// TIA Portal V16 export
// export: Created 2021-11-12T13:32:39.4963653Z, ExportSetting WithDefaults, DisplayName Totally Integrated Automation Portal, DisplayVersion V16 Update 3, DisplayName TIA Portal Version Control Interface, DisplayVersion V16 Update 2, DisplayName TIA Portal Openness, DisplayVersion V16 Update 3, DisplayName SINAMICS Startdrive Advanced, DisplayVersion V16 Update 5, DisplayName SINAMICS Startdrive G130, G150, S120, S150, SINAMICS MV, S210, DisplayVersion V16 Update 5, DisplayName SINAMICS Startdrive G110M, G120, G120C, G120D, G120P, G115D, DisplayVersion V16 Update 5, DisplayName STEP 7 Professional, DisplayVersion V16 Update 3, DisplayName STEP 7 Safety, DisplayVersion V16, DisplayName WinCC UA Professional, DisplayVersion V16 Update 3
FUNCTION_BLOCK "Station2R2"   // FB19, LAD
{ S7_Optimized_Access := 'TRUE' }
VERSION : 0.1
// stored: AutoNumber true, IsIECCheckEnabled false, IsRetainMemResEnabled false, MemoryReserve 100, SetENOAutomatically false, UDAEnableTagReadback false
   VAR
      SF_RO01_Timeout : "STD_DI_Mon";
      SF_RO01_LubStartErr { S7_SetPoint := 'True'} : "STD_DI_Mon";
      "SF_CM01-BL01_Wrn" { S7_SetPoint := 'True'} : "STD_DI_Mon";
      "SF_CM01-BL01_Err" { S7_SetPoint := 'True'} : "STD_DI_Mon";
      SF_RO01 { S7_SetPoint := 'True'} : "STD_RobotABB";
      SF_RC01 : "STD_DriveRobotABB";
      SS_Edge { S7_SetPoint := 'True'} : Array[0..16] of Bool;
      SB1ReqServPos { ExternalAccessible := 'False'; ExternalVisible := 'False'; ExternalWritable := 'False'} : Bool;   // Request to go to/from service position
      SB1ReqToolchange : Bool;   // Go to position for change tool request
      SB1ReqFlush : Bool;   // Request to flash tool
      SB1ReqFlushAux { ExternalAccessible := 'False'; ExternalVisible := 'False'; ExternalWritable := 'False'} : Bool;   // Manual (HW button) request to flush
      SB1ReqSprayMan : Bool;   // Manual (HW button) request to spray
      SB1ReqSprayManAux { ExternalAccessible := 'False'; ExternalVisible := 'False'; ExternalWritable := 'False'} : Bool;   // Manual (HW button) request to spray
      SB1CycleAutostop : Bool;   // Cycle autostop command
      SB1RobotInitialized : Bool;   // SB1RobotInitialized
   END_VAR
   VAR_TEMP
      TS_RC01 : "UDT_DriveRobotABBControl";   // Robot RO01 control
      TS_RO01 : "UDT_RobotABBControl";   // Robot RO01 control
      TB1PwrOK : Bool;   // Power for this station is OK
      TB1CtrlRun : Bool;   // Robot controller is running in automat
      TB1HomePos : Bool;   // Request to go to home position
      TB1MoveOutPress : Bool;   // Move robout out of press
      TB1SprayInPress : Bool;   // Spray into press
      TB1SprayOutPress : Bool;   // Spray out off press
      TB1SprayMan : Bool;   // Spray manually both ways
      TB1Flush : Bool;   // Flush tool
      TB1MoveToStandBy : Bool;   // From home to StandBy
      TB1PressFree : Bool;   // positions in press are free
      TB1PartsBefore : Bool;   // Parts in zone before robot
   END_VAR
   VAR CONSTANT
      CI_JobHome : UInt := 1;   // Go home
      CI_JobService : UInt := 2;   // Go service
      CI_JobToolchange : UInt := 3;   // Go to position for change tool
      CI_JobMoveOutPress : UInt := 11;   // Move out of the press
      CI_JobStandBy : UInt := 12;   // From home to StandBy
      CI_JobSprayIntoPress : UInt := 101;   // Spray into the press
      CI_JobSprayOutPress : UInt := 102;   // Spray out of the press
      CI_JobSprayMan : UInt := 110;   // Spray manually both ways
      CI_JobFlushTool : UInt := 200;   // Flush
   END_VAR
   VAR_TEMP   // added for the SCL form of the ladder/FBD networks
      _w1 : Bool;
      _w2 : Bool;
      _w3 : Bool;
      _w4 : Bool;
   END_VAR
BEGIN

REGION Network 1: Clear temporary variables
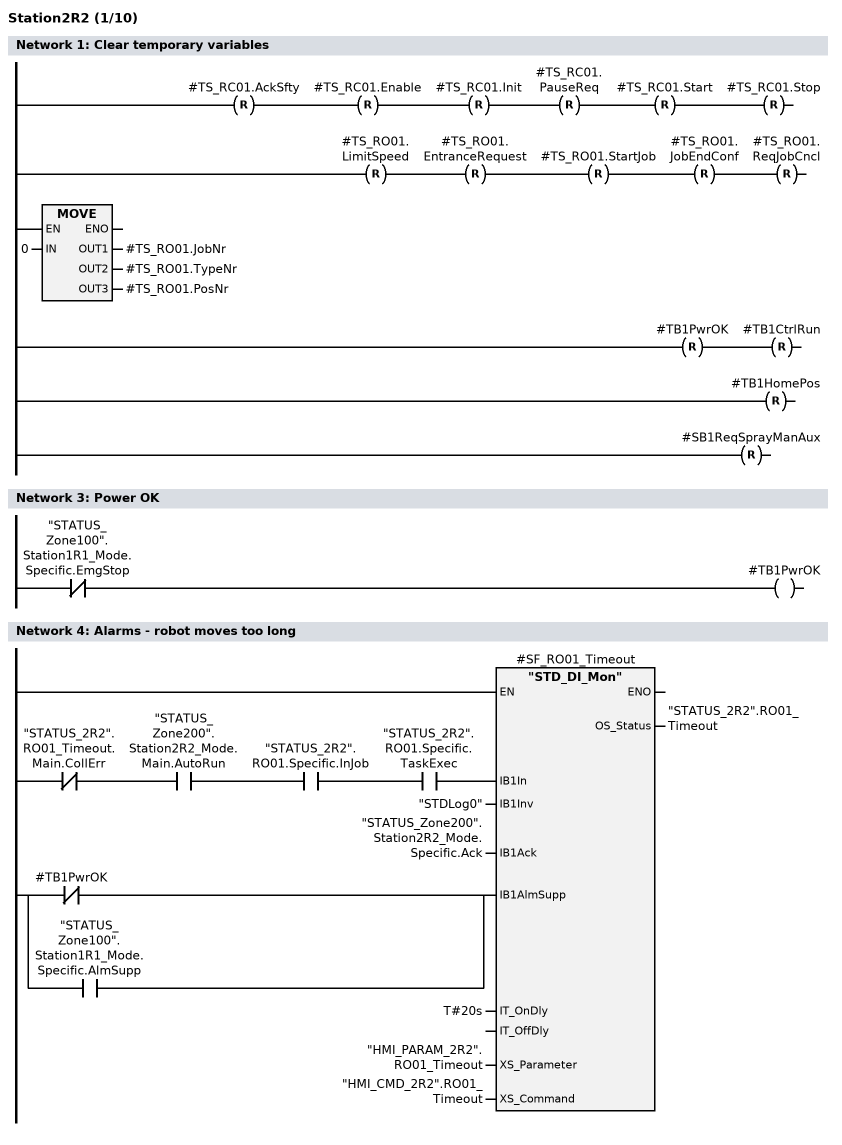
   RUNG wire#powerrail
      R_Coil( #TS_RC01.AckSfty )
      R_Coil( #TS_RC01.Enable )
      R_Coil( #TS_RC01.Init )
      R_Coil( #TS_RC01.PauseReq )
      R_Coil( #TS_RC01.Start )
      R_Coil( #TS_RC01.Stop )
   END_RUNG
   RUNG wire#powerrail
      R_Coil( #TS_RO01.LimitSpeed )
      R_Coil( #TS_RO01.EntranceRequest )
      R_Coil( #TS_RO01.StartJob )
      R_Coil( #TS_RO01.JobEndConf )
      R_Coil( #TS_RO01.ReqJobCncl )
   END_RUNG
   RUNG wire#powerrail
      Move(in := 0, out1 => #TS_RO01.JobNr, out2 => #TS_RO01.TypeNr, out3 => #TS_RO01.PosNr)
   END_RUNG
   RUNG wire#powerrail
      R_Coil( #TB1PwrOK )
      R_Coil( #TB1CtrlRun )
   END_RUNG
   RUNG wire#powerrail
      R_Coil( #TB1HomePos )
   END_RUNG
   RUNG wire#powerrail
      R_Coil( #SB1ReqSprayManAux )
   END_RUNG
   // the same network as SCL:
   #TS_RC01.AckSfty := FALSE;
   #TS_RC01.Enable := FALSE;
   #TS_RC01.Init := FALSE;
   #TS_RC01.PauseReq := FALSE;
   #TS_RC01.Start := FALSE;
   #TS_RC01.Stop := FALSE;
   #TS_RO01.LimitSpeed := FALSE;
   #TS_RO01.EntranceRequest := FALSE;
   #TS_RO01.StartJob := FALSE;
   #TS_RO01.JobEndConf := FALSE;
   #TS_RO01.ReqJobCncl := FALSE;
   #TS_RO01.JobNr := 0;
   #TS_RO01.TypeNr := 0;
   #TS_RO01.PosNr := 0;
   #TB1PwrOK := FALSE;
   #TB1CtrlRun := FALSE;
   #TB1HomePos := FALSE;
   #SB1ReqSprayManAux := FALSE;
END_REGION

REGION Network 2: *************** Alarms ***************
END_REGION

REGION Network 3: Power OK
   RUNG wire#powerrail
      I_Contact( "STATUS_Zone100".Station1R1_Mode.Specific.EmgStop )
      Coil( #TB1PwrOK )
   END_RUNG
   // the same network as SCL:
   #TB1PwrOK := NOT "STATUS_Zone100".Station1R1_Mode.Specific.EmgStop;
END_REGION

REGION Network 4: Alarms - robot moves too long
   RUNG wire#powerrail
      #SF_RO01_Timeout(IB1In := wire#w1, IB1AlmSupp := wire#w2, IB1Inv := "STDLog0", IB1Ack := "STATUS_Zone200".Station2R2_Mode.Specific.Ack, IT_OnDly := T#20s, IT_OffDly :=, XS_Parameter := "HMI_PARAM_2R2".RO01_Timeout, XS_Command := "HMI_CMD_2R2".RO01_Timeout, OS_Status => "STATUS_2R2".RO01_Timeout)
   END_RUNG
   RUNG wire#powerrail
      I_Contact( "STATUS_2R2".RO01_Timeout.Main.CollErr )
      Contact( "STATUS_Zone200".Station2R2_Mode.Main.AutoRun )
      Contact( "STATUS_2R2".RO01.Specific.InJob )
      Contact( "STATUS_2R2".RO01.Specific.TaskExec )
   END_RUNG wire#w1
   RUNG wire#powerrail
      I_Contact( #TB1PwrOK )
   END_RUNG wire#w2
   RUNG wire#powerrail
      Contact( "STATUS_Zone100".Station1R1_Mode.Specific.AlmSupp )
   END_RUNG wire#w2
   // the same network as SCL:
   #SF_RO01_Timeout(IB1In := NOT "STATUS_2R2".RO01_Timeout.Main.CollErr AND "STATUS_Zone200".Station2R2_Mode.Main.AutoRun AND "STATUS_2R2".RO01.Specific.InJob AND "STATUS_2R2".RO01.Specific.TaskExec,   // "STD_DI_Mon"
                    IB1Inv := "STDLog0",
                    IB1Ack := "STATUS_Zone200".Station2R2_Mode.Specific.Ack,
                    IB1AlmSupp := NOT #TB1PwrOK OR "STATUS_Zone100".Station1R1_Mode.Specific.AlmSupp,
                    IT_OnDly := T#20s,
                    XS_Parameter := "HMI_PARAM_2R2".RO01_Timeout,
                    XS_Command := "HMI_CMD_2R2".RO01_Timeout,
                    OS_Status => "STATUS_2R2".RO01_Timeout);
END_REGION

REGION Network 5: Alarm - robot did not move into the press machine
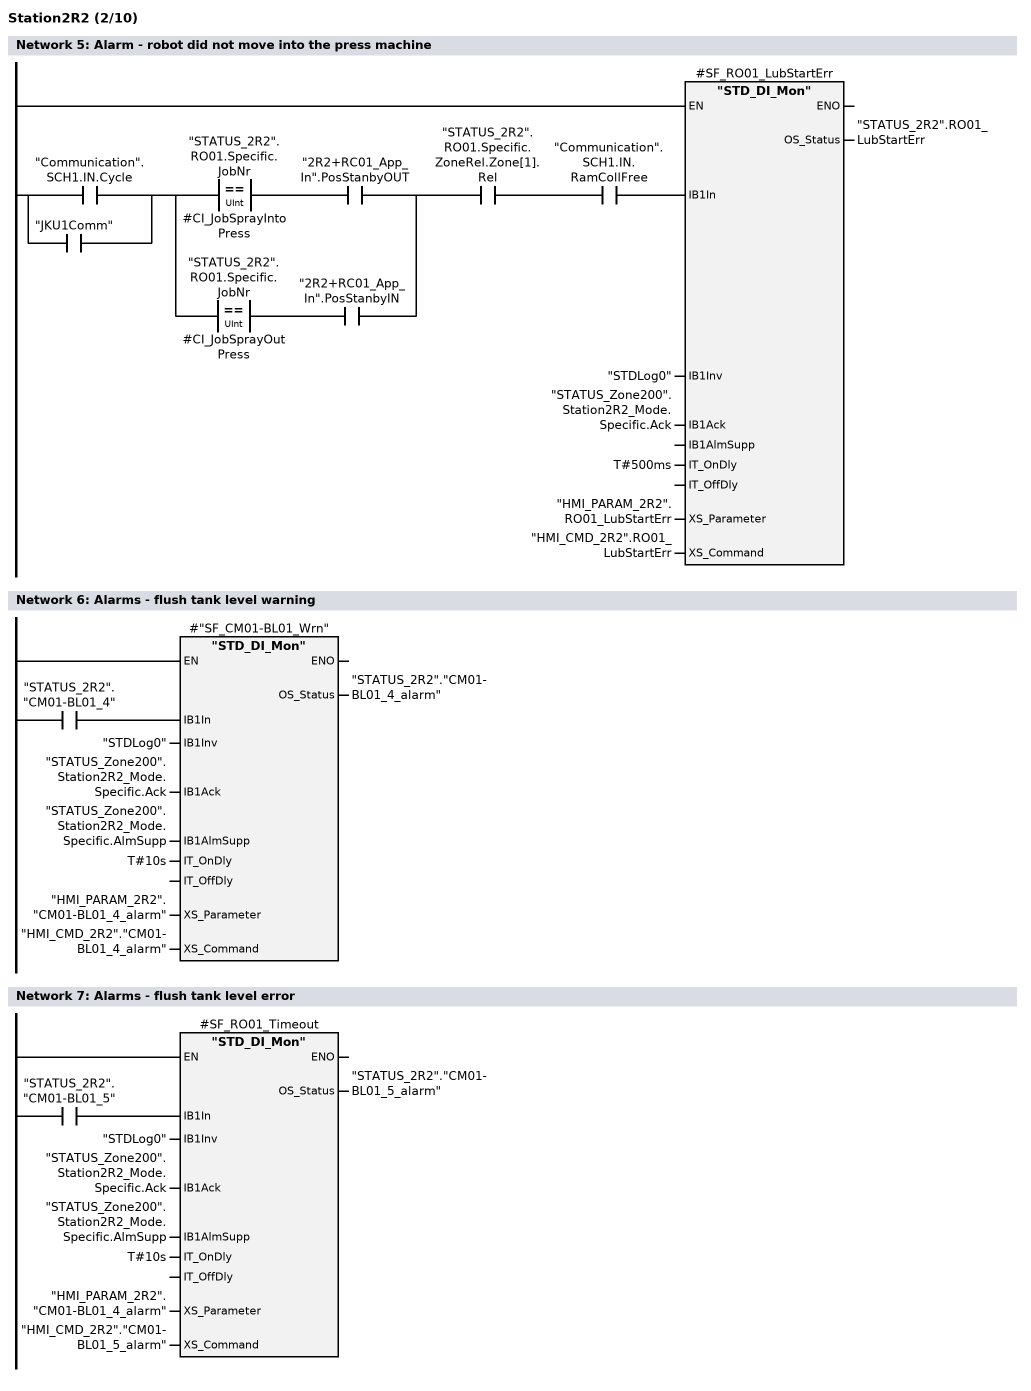
   RUNG wire#powerrail
      #SF_RO01_LubStartErr(IB1In := wire#w3, IB1Inv := "STDLog0", IB1Ack := "STATUS_Zone200".Station2R2_Mode.Specific.Ack, IB1AlmSupp :=, IT_OnDly := T#500ms, IT_OffDly :=, XS_Parameter := "HMI_PARAM_2R2".RO01_LubStartErr, XS_Command := "HMI_CMD_2R2".RO01_LubStartErr, OS_Status => "STATUS_2R2".RO01_LubStartErr)
   END_RUNG
   RUNG wire#powerrail
      Contact( "Communication".SCH1.IN.Cycle )
      wire#w1
      { S7_Templates := "SrcType := UInt" } EQ_Contact(in1 := "STATUS_2R2".RO01.Specific.JobNr, in2 := #CI_JobSprayIntoPress)
      Contact( "2R2+RC01_App_In".PosStanbyOUT )
      wire#w2
      Contact( "STATUS_2R2".RO01.Specific.ZoneRel.Zone[1].Rel )
      Contact( "Communication".SCH1.IN.RamCollFree )
   END_RUNG wire#w3
   RUNG wire#powerrail
      Contact( "JKU1Comm" )
   END_RUNG wire#w1
   RUNG wire#w1
      { S7_Templates := "SrcType := UInt" } EQ_Contact(in1 := "STATUS_2R2".RO01.Specific.JobNr, in2 := #CI_JobSprayOutPress)
      Contact( "2R2+RC01_App_In".PosStanbyIN )
   END_RUNG wire#w2
   // the same network as SCL:
   #SF_RO01_LubStartErr(IB1In := ("Communication".SCH1.IN.Cycle OR "JKU1Comm") AND ((("STATUS_2R2".RO01.Specific.JobNr = #CI_JobSprayIntoPress) AND "2R2+RC01_App_In".PosStanbyOUT) OR (("STATUS_2R2".RO01.Specific.JobNr = #CI_JobSprayOutPress) AND "2R2+RC01_App_In".PosStanbyIN)) AND "STATUS_2R2".RO01.Specific.ZoneRel.Zone[1].Rel AND "Communication".SCH1.IN.RamCollFree,   // "STD_DI_Mon"
                        IB1Inv := "STDLog0",
                        IB1Ack := "STATUS_Zone200".Station2R2_Mode.Specific.Ack,
                        IT_OnDly := T#500ms,
                        XS_Parameter := "HMI_PARAM_2R2".RO01_LubStartErr,
                        XS_Command := "HMI_CMD_2R2".RO01_LubStartErr,
                        OS_Status => "STATUS_2R2".RO01_LubStartErr);
END_REGION

REGION Network 6: Alarms - flush tank level warning
   RUNG wire#powerrail
      #"SF_CM01-BL01_Wrn"(IB1In := wire#w1, IB1Inv := "STDLog0", IB1Ack := "STATUS_Zone200".Station2R2_Mode.Specific.Ack, IB1AlmSupp := "STATUS_Zone200".Station2R2_Mode.Specific.AlmSupp, IT_OnDly := T#10s, IT_OffDly :=, XS_Parameter := "HMI_PARAM_2R2"."CM01-BL01_4_alarm", XS_Command := "HMI_CMD_2R2"."CM01-BL01_4_alarm", OS_Status => "STATUS_2R2"."CM01-BL01_4_alarm")
   END_RUNG
   RUNG wire#powerrail
      Contact( "STATUS_2R2"."CM01-BL01_4" )
   END_RUNG wire#w1
   // the same network as SCL:
   #"SF_CM01-BL01_Wrn"(IB1In := "STATUS_2R2"."CM01-BL01_4",   // "STD_DI_Mon"
                       IB1Inv := "STDLog0",
                       IB1Ack := "STATUS_Zone200".Station2R2_Mode.Specific.Ack,
                       IB1AlmSupp := "STATUS_Zone200".Station2R2_Mode.Specific.AlmSupp,
                       IT_OnDly := T#10s,
                       XS_Parameter := "HMI_PARAM_2R2"."CM01-BL01_4_alarm",
                       XS_Command := "HMI_CMD_2R2"."CM01-BL01_4_alarm",
                       OS_Status => "STATUS_2R2"."CM01-BL01_4_alarm");
END_REGION

REGION Network 7: Alarms - flush tank level error
   RUNG wire#powerrail
      #SF_RO01_Timeout(IB1In := wire#w1, IB1Inv := "STDLog0", IB1Ack := "STATUS_Zone200".Station2R2_Mode.Specific.Ack, IB1AlmSupp := "STATUS_Zone200".Station2R2_Mode.Specific.AlmSupp, IT_OnDly := T#10s, IT_OffDly :=, XS_Parameter := "HMI_PARAM_2R2"."CM01-BL01_4_alarm", XS_Command := "HMI_CMD_2R2"."CM01-BL01_5_alarm", OS_Status => "STATUS_2R2"."CM01-BL01_5_alarm")
   END_RUNG
   RUNG wire#powerrail
      Contact( "STATUS_2R2"."CM01-BL01_5" )
   END_RUNG wire#w1
   // the same network as SCL:
   #SF_RO01_Timeout(IB1In := "STATUS_2R2"."CM01-BL01_5",   // "STD_DI_Mon"
                    IB1Inv := "STDLog0",
                    IB1Ack := "STATUS_Zone200".Station2R2_Mode.Specific.Ack,
                    IB1AlmSupp := "STATUS_Zone200".Station2R2_Mode.Specific.AlmSupp,
                    IT_OnDly := T#10s,
                    XS_Parameter := "HMI_PARAM_2R2"."CM01-BL01_4_alarm",
                    XS_Command := "HMI_CMD_2R2"."CM01-BL01_5_alarm",
                    OS_Status => "STATUS_2R2"."CM01-BL01_5_alarm");
END_REGION

REGION Network 8: *************** Controller RC01 ***************
END_REGION

REGION Network 9: RC01 - control
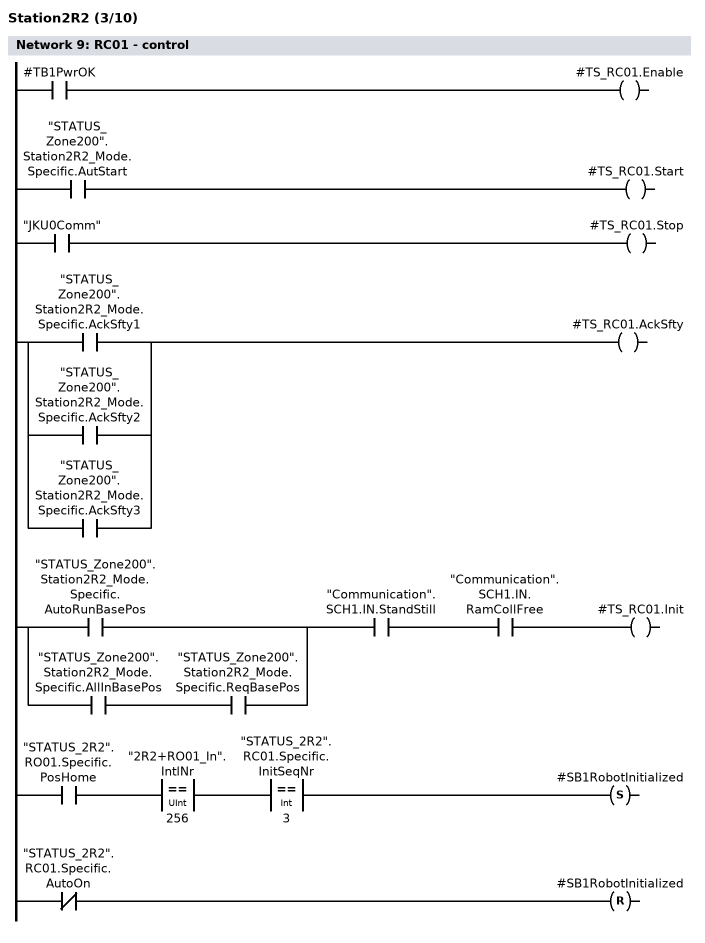
   RUNG wire#powerrail
      Contact( #TB1PwrOK )
      Coil( #TS_RC01.Enable )
   END_RUNG
   RUNG wire#powerrail
      Contact( "STATUS_Zone200".Station2R2_Mode.Specific.AutStart )
      Coil( #TS_RC01.Start )
   END_RUNG
   RUNG wire#powerrail
      Contact( "JKU0Comm" )
      Coil( #TS_RC01.Stop )
   END_RUNG
   RUNG wire#powerrail
      Contact( "STATUS_Zone200".Station2R2_Mode.Specific.AckSfty1 )
      wire#w1
      Coil( #TS_RC01.AckSfty )
   END_RUNG
   RUNG wire#powerrail
      Contact( "STATUS_Zone200".Station2R2_Mode.Specific.AckSfty2 )
   END_RUNG wire#w1
   RUNG wire#powerrail
      Contact( "STATUS_Zone200".Station2R2_Mode.Specific.AckSfty3 )
   END_RUNG wire#w1
   RUNG wire#powerrail
      Contact( "STATUS_Zone200".Station2R2_Mode.Specific.AutoRunBasePos )
      wire#w2
      Contact( "Communication".SCH1.IN.StandStill )
      Contact( "Communication".SCH1.IN.RamCollFree )
      Coil( #TS_RC01.Init )
   END_RUNG
   RUNG wire#powerrail
      Contact( "STATUS_Zone200".Station2R2_Mode.Specific.AllInBasePos )
      Contact( "STATUS_Zone200".Station2R2_Mode.Specific.ReqBasePos )
   END_RUNG wire#w2
   RUNG wire#powerrail
      Contact( "STATUS_2R2".RO01.Specific.PosHome )
      { S7_Templates := "SrcType := UInt" } EQ_Contact(in1 := "2R2+RO01_In".IntlNr, in2 := 256)
      { S7_Templates := "SrcType := Int" } EQ_Contact(in1 := "STATUS_2R2".RC01.Specific.InitSeqNr, in2 := 3)
      S_Coil( #SB1RobotInitialized )
   END_RUNG
   RUNG wire#powerrail
      I_Contact( "STATUS_2R2".RC01.Specific.AutoOn )
      R_Coil( #SB1RobotInitialized )
   END_RUNG
   // the same network as SCL:
   #TS_RC01.Enable := #TB1PwrOK;
   #TS_RC01.Start := "STATUS_Zone200".Station2R2_Mode.Specific.AutStart;
   #TS_RC01.Stop := "JKU0Comm";
   #TS_RC01.AckSfty := "STATUS_Zone200".Station2R2_Mode.Specific.AckSfty1 OR "STATUS_Zone200".Station2R2_Mode.Specific.AckSfty2 OR "STATUS_Zone200".Station2R2_Mode.Specific.AckSfty3;
   #TS_RC01.Init := ("STATUS_Zone200".Station2R2_Mode.Specific.AutoRunBasePos OR ("STATUS_Zone200".Station2R2_Mode.Specific.AllInBasePos AND "STATUS_Zone200".Station2R2_Mode.Specific.ReqBasePos)) AND "Communication".SCH1.IN.StandStill AND "Communication".SCH1.IN.RamCollFree;
   IF "STATUS_2R2".RO01.Specific.PosHome AND ("2R2+RO01_In".IntlNr = 256) AND ("STATUS_2R2".RC01.Specific.InitSeqNr = 3) THEN
       #SB1RobotInitialized := TRUE;
   END_IF;
   IF NOT "STATUS_2R2".RC01.Specific.AutoOn THEN #SB1RobotInitialized := FALSE; END_IF;
END_REGION

REGION Network 10: RC01 - request to pause robots jobs
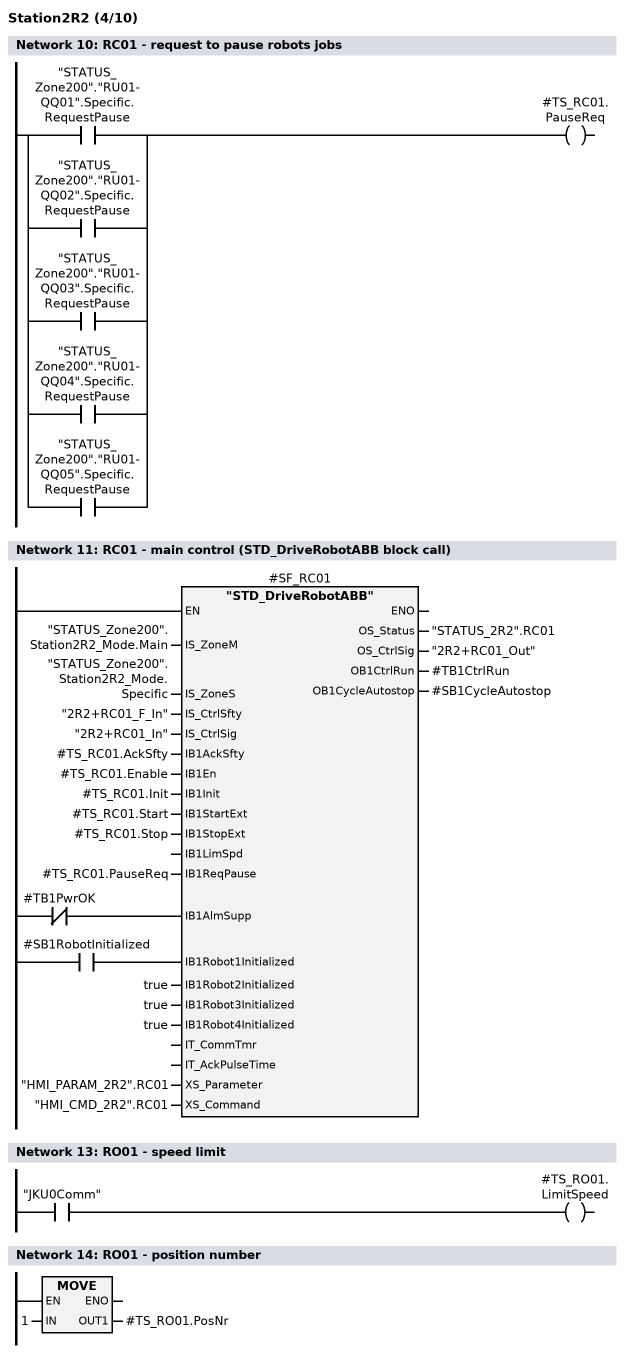
   RUNG wire#powerrail
      Contact( "STATUS_Zone200"."RU01-QQ01".Specific.RequestPause )
      wire#w1
      Coil( #TS_RC01.PauseReq )
   END_RUNG
   RUNG wire#powerrail
      Contact( "STATUS_Zone200"."RU01-QQ02".Specific.RequestPause )
   END_RUNG wire#w1
   RUNG wire#powerrail
      Contact( "STATUS_Zone200"."RU01-QQ03".Specific.RequestPause )
   END_RUNG wire#w1
   RUNG wire#powerrail
      Contact( "STATUS_Zone200"."RU01-QQ04".Specific.RequestPause )
   END_RUNG wire#w1
   RUNG wire#powerrail
      Contact( "STATUS_Zone200"."RU01-QQ05".Specific.RequestPause )
   END_RUNG wire#w1
   // the same network as SCL:
   #TS_RC01.PauseReq := "STATUS_Zone200"."RU01-QQ01".Specific.RequestPause OR "STATUS_Zone200"."RU01-QQ02".Specific.RequestPause OR "STATUS_Zone200"."RU01-QQ03".Specific.RequestPause OR "STATUS_Zone200"."RU01-QQ04".Specific.RequestPause OR "STATUS_Zone200"."RU01-QQ05".Specific.RequestPause;
END_REGION

REGION Network 11: RC01 - main control (STD_DriveRobotABB block call)
   RUNG wire#powerrail
      #SF_RC01(IB1AlmSupp := wire#w1, IB1Robot1Initialized := wire#w2, IS_ZoneM := "STATUS_Zone200".Station2R2_Mode.Main, IS_ZoneS := "STATUS_Zone200".Station2R2_Mode.Specific, IS_CtrlSfty := "2R2+RC01_F_In", IS_CtrlSig := "2R2+RC01_In", IB1AckSfty := #TS_RC01.AckSfty, IB1En := #TS_RC01.Enable, IB1Init := #TS_RC01.Init, IB1StartExt := #TS_RC01.Start, IB1StopExt := #TS_RC01.Stop, IB1LimSpd :=, IB1ReqPause := #TS_RC01.PauseReq, IB1Robot2Initialized := true, IB1Robot3Initialized := true, IB1Robot4Initialized := true, IT_CommTmr :=, IT_AckPulseTime :=, XS_Parameter := "HMI_PARAM_2R2".RC01, XS_Command := "HMI_CMD_2R2".RC01, OS_Status => "STATUS_2R2".RC01, OS_CtrlSig => "2R2+RC01_Out", OB1CtrlRun => #TB1CtrlRun, OB1CycleAutostop => #SB1CycleAutostop)
   END_RUNG
   RUNG wire#powerrail
      I_Contact( #TB1PwrOK )
   END_RUNG wire#w1
   RUNG wire#powerrail
      Contact( #SB1RobotInitialized )
   END_RUNG wire#w2
   // the same network as SCL:
   #SF_RC01(IS_ZoneM := "STATUS_Zone200".Station2R2_Mode.Main,   // "STD_DriveRobotABB"
            IS_ZoneS := "STATUS_Zone200".Station2R2_Mode.Specific,
            IS_CtrlSfty := "2R2+RC01_F_In",
            IS_CtrlSig := "2R2+RC01_In",
            IB1AckSfty := #TS_RC01.AckSfty,
            IB1En := #TS_RC01.Enable,
            IB1Init := #TS_RC01.Init,
            IB1StartExt := #TS_RC01.Start,
            IB1StopExt := #TS_RC01.Stop,
            IB1ReqPause := #TS_RC01.PauseReq,
            IB1AlmSupp := NOT #TB1PwrOK,
            IB1Robot1Initialized := #SB1RobotInitialized,
            IB1Robot2Initialized := true,
            IB1Robot3Initialized := true,
            IB1Robot4Initialized := true,
            XS_Parameter := "HMI_PARAM_2R2".RC01,
            XS_Command := "HMI_CMD_2R2".RC01,
            OS_Status => "STATUS_2R2".RC01,
            OS_CtrlSig => "2R2+RC01_Out",
            OB1CtrlRun => #TB1CtrlRun,
            OB1CycleAutostop => #SB1CycleAutostop);
END_REGION

REGION Network 12: *************** Robot RO01 ***************
END_REGION

REGION Network 13: RO01 - speed limit
   RUNG wire#powerrail
      Contact( "JKU0Comm" )
      Coil( #TS_RO01.LimitSpeed )
   END_RUNG
   // the same network as SCL:
   #TS_RO01.LimitSpeed := "JKU0Comm";
END_REGION

REGION Network 14: RO01 - position number
   RUNG wire#powerrail
      Move(in := 1, out1 => #TS_RO01.PosNr)
   END_RUNG
   // the same network as SCL:
   #TS_RO01.PosNr := 1;
END_REGION

REGION Network 15: RO01 - confirm end of job
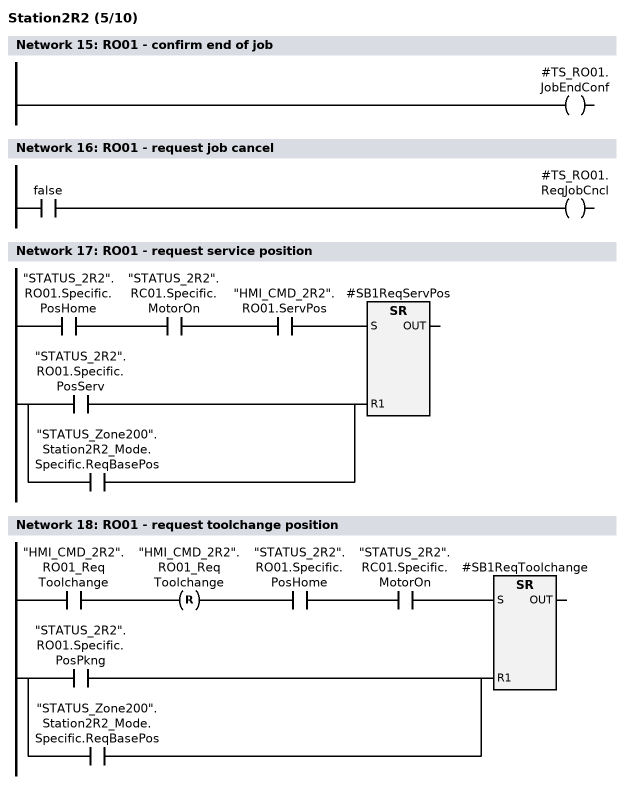
   RUNG wire#powerrail
      Coil( #TS_RO01.JobEndConf )
   END_RUNG
   // the same network as SCL:
   #TS_RO01.JobEndConf := TRUE;
END_REGION

REGION Network 16: RO01 - request job cancel
   RUNG wire#powerrail
      Contact( false )
      Coil( #TS_RO01.ReqJobCncl )
   END_RUNG
   // the same network as SCL:
   #TS_RO01.ReqJobCncl := false;
END_REGION

REGION Network 17: RO01 - request service position
   RUNG wire#powerrail
      Contact( "STATUS_2R2".RO01.Specific.PosHome )
      Contact( "STATUS_2R2".RC01.Specific.MotorOn )
      Contact( "HMI_CMD_2R2".RO01.ServPos )
      S_SR(operand := #SB1ReqServPos, r1 := wire#w1)
   END_RUNG
   RUNG wire#powerrail
      Contact( "STATUS_2R2".RO01.Specific.PosServ )
   END_RUNG wire#w1
   RUNG wire#powerrail
      Contact( "STATUS_Zone200".Station2R2_Mode.Specific.ReqBasePos )
   END_RUNG wire#w1
   // the same network as SCL:
   IF "STATUS_2R2".RO01.Specific.PosHome AND "STATUS_2R2".RC01.Specific.MotorOn AND "HMI_CMD_2R2".RO01.ServPos THEN
       #SB1ReqServPos := TRUE;   // SR flip-flop
   END_IF;
   IF "STATUS_2R2".RO01.Specific.PosServ OR "STATUS_Zone200".Station2R2_Mode.Specific.ReqBasePos THEN
       #SB1ReqServPos := FALSE;
   END_IF;
END_REGION

REGION Network 18: RO01 - request toolchange position
   RUNG wire#powerrail
      Contact( "HMI_CMD_2R2".RO01_ReqToolchange )
      R_Coil( "HMI_CMD_2R2".RO01_ReqToolchange )
      Contact( "STATUS_2R2".RO01.Specific.PosHome )
      Contact( "STATUS_2R2".RC01.Specific.MotorOn )
      S_SR(operand := #SB1ReqToolchange, r1 := wire#w1)
   END_RUNG
   RUNG wire#powerrail
      Contact( "STATUS_2R2".RO01.Specific.PosPkng )
   END_RUNG wire#w1
   RUNG wire#powerrail
      Contact( "STATUS_Zone200".Station2R2_Mode.Specific.ReqBasePos )
   END_RUNG wire#w1
   // the same network as SCL:
   #_w1 := "HMI_CMD_2R2".RO01_ReqToolchange;
   IF #_w1 THEN "HMI_CMD_2R2".RO01_ReqToolchange := FALSE; END_IF;
   IF #_w1 AND "STATUS_2R2".RO01.Specific.PosHome AND "STATUS_2R2".RC01.Specific.MotorOn THEN
       #SB1ReqToolchange := TRUE;   // SR flip-flop
   END_IF;
   IF "STATUS_2R2".RO01.Specific.PosPkng OR "STATUS_Zone200".Station2R2_Mode.Specific.ReqBasePos THEN
       #SB1ReqToolchange := FALSE;
   END_IF;
END_REGION

REGION Network 19: Parts in zone before robot
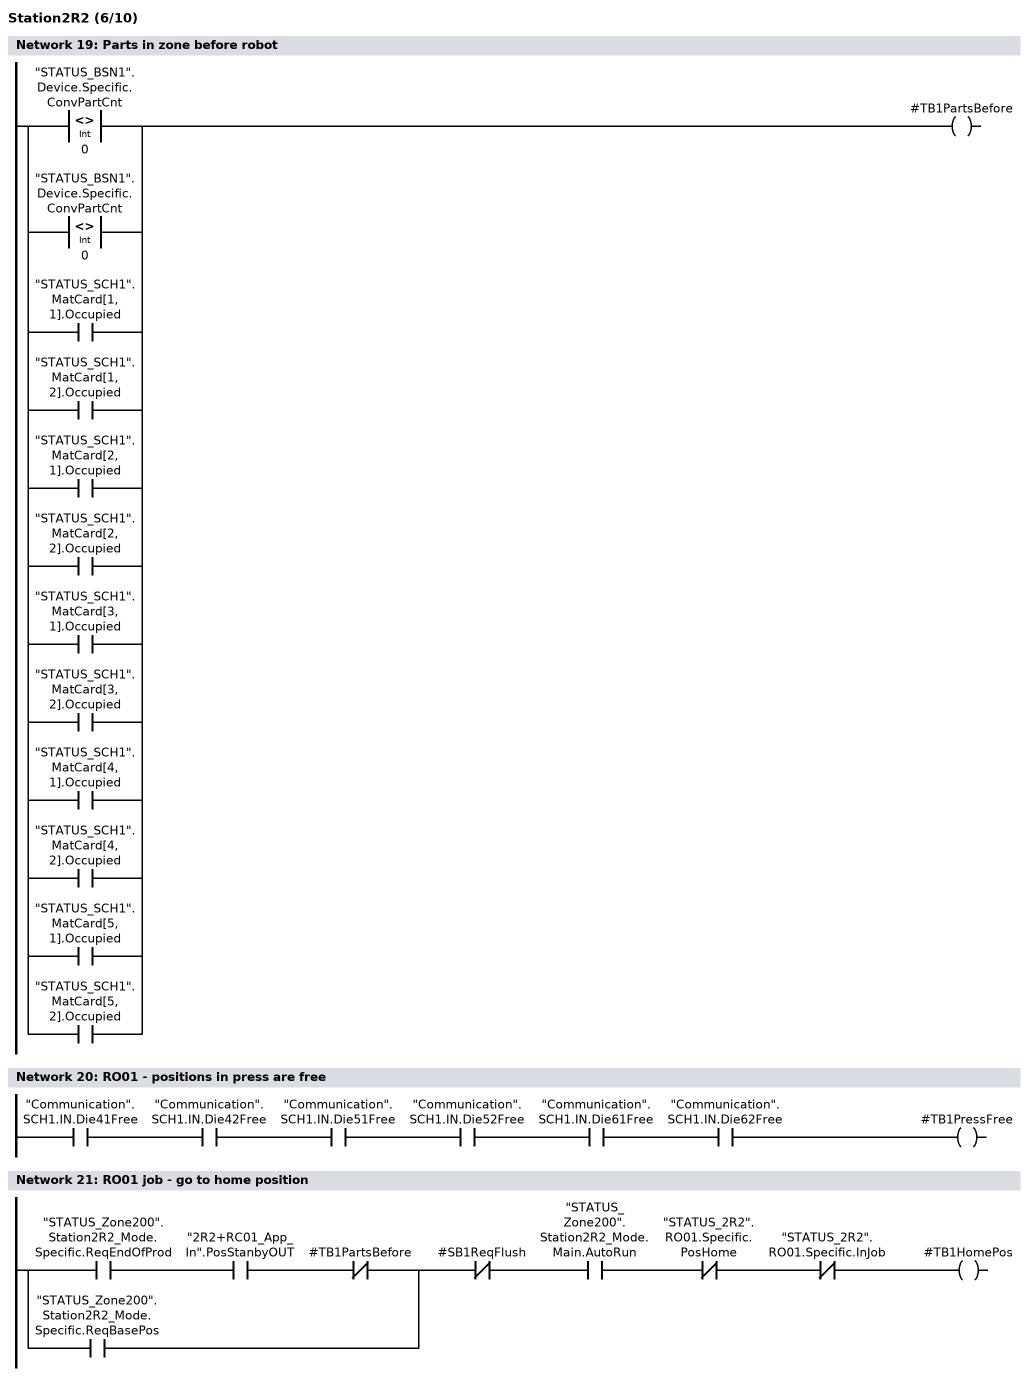
   RUNG wire#powerrail
      { S7_Templates := "SrcType := Int" } NE_Contact(in1 := "STATUS_BSN1".Device.Specific.ConvPartCnt, in2 := 0)
      wire#w1
      Coil( #TB1PartsBefore )
   END_RUNG
   RUNG wire#powerrail
      { S7_Templates := "SrcType := Int" } NE_Contact(in1 := "STATUS_BSN1".Device.Specific.ConvPartCnt, in2 := 0)
   END_RUNG wire#w1
   RUNG wire#powerrail
      Contact( "STATUS_SCH1".MatCard[1, 1].Occupied )
   END_RUNG wire#w1
   RUNG wire#powerrail
      Contact( "STATUS_SCH1".MatCard[1, 2].Occupied )
   END_RUNG wire#w1
   RUNG wire#powerrail
      Contact( "STATUS_SCH1".MatCard[2, 1].Occupied )
   END_RUNG wire#w1
   RUNG wire#powerrail
      Contact( "STATUS_SCH1".MatCard[2, 2].Occupied )
   END_RUNG wire#w1
   RUNG wire#powerrail
      Contact( "STATUS_SCH1".MatCard[3, 1].Occupied )
   END_RUNG wire#w1
   RUNG wire#powerrail
      Contact( "STATUS_SCH1".MatCard[3, 2].Occupied )
   END_RUNG wire#w1
   RUNG wire#powerrail
      Contact( "STATUS_SCH1".MatCard[4, 1].Occupied )
   END_RUNG wire#w1
   RUNG wire#powerrail
      Contact( "STATUS_SCH1".MatCard[4, 2].Occupied )
   END_RUNG wire#w1
   RUNG wire#powerrail
      Contact( "STATUS_SCH1".MatCard[5, 1].Occupied )
   END_RUNG wire#w1
   RUNG wire#powerrail
      Contact( "STATUS_SCH1".MatCard[5, 2].Occupied )
   END_RUNG wire#w1
   // the same network as SCL:
   #TB1PartsBefore := ("STATUS_BSN1".Device.Specific.ConvPartCnt <> 0) OR ("STATUS_BSN1".Device.Specific.ConvPartCnt <> 0) OR "STATUS_SCH1".MatCard[1, 1].Occupied OR "STATUS_SCH1".MatCard[1, 2].Occupied OR "STATUS_SCH1".MatCard[2, 1].Occupied OR "STATUS_SCH1".MatCard[2, 2].Occupied OR "STATUS_SCH1".MatCard[3, 1].Occupied OR "STATUS_SCH1".MatCard[3, 2].Occupied OR "STATUS_SCH1".MatCard[4, 1].Occupied OR "STATUS_SCH1".MatCard[4, 2].Occupied OR "STATUS_SCH1".MatCard[5, 1].Occupied OR "STATUS_SCH1".MatCard[5, 2].Occupied;
END_REGION

REGION Network 20: RO01 - positions in press are free
   RUNG wire#powerrail
      Contact( "Communication".SCH1.IN.Die41Free )
      Contact( "Communication".SCH1.IN.Die42Free )
      Contact( "Communication".SCH1.IN.Die51Free )
      Contact( "Communication".SCH1.IN.Die52Free )
      Contact( "Communication".SCH1.IN.Die61Free )
      Contact( "Communication".SCH1.IN.Die62Free )
      Coil( #TB1PressFree )
   END_RUNG
   // the same network as SCL:
   #TB1PressFree := "Communication".SCH1.IN.Die41Free AND "Communication".SCH1.IN.Die42Free AND "Communication".SCH1.IN.Die51Free AND "Communication".SCH1.IN.Die52Free AND "Communication".SCH1.IN.Die61Free AND "Communication".SCH1.IN.Die62Free;
END_REGION

REGION Network 21: RO01 job - go to home position
   RUNG wire#powerrail
      Contact( "STATUS_Zone200".Station2R2_Mode.Specific.ReqEndOfProd )
      Contact( "2R2+RC01_App_In".PosStanbyOUT )
      I_Contact( #TB1PartsBefore )
      wire#w1
      I_Contact( #SB1ReqFlush )
      Contact( "STATUS_Zone200".Station2R2_Mode.Main.AutoRun )
      I_Contact( "STATUS_2R2".RO01.Specific.PosHome )
      I_Contact( "STATUS_2R2".RO01.Specific.InJob )
      Coil( #TB1HomePos )
   END_RUNG
   RUNG wire#powerrail
      Contact( "STATUS_Zone200".Station2R2_Mode.Specific.ReqBasePos )
   END_RUNG wire#w1
   // the same network as SCL:
   #TB1HomePos := (("STATUS_Zone200".Station2R2_Mode.Specific.ReqEndOfProd AND "2R2+RC01_App_In".PosStanbyOUT AND NOT #TB1PartsBefore) OR "STATUS_Zone200".Station2R2_Mode.Specific.ReqBasePos) AND NOT #SB1ReqFlush AND "STATUS_Zone200".Station2R2_Mode.Main.AutoRun AND NOT "STATUS_2R2".RO01.Specific.PosHome AND NOT "STATUS_2R2".RO01.Specific.InJob;
END_REGION

REGION Network 22: RO01 job - go to standby position (from home to in front of the press machine)
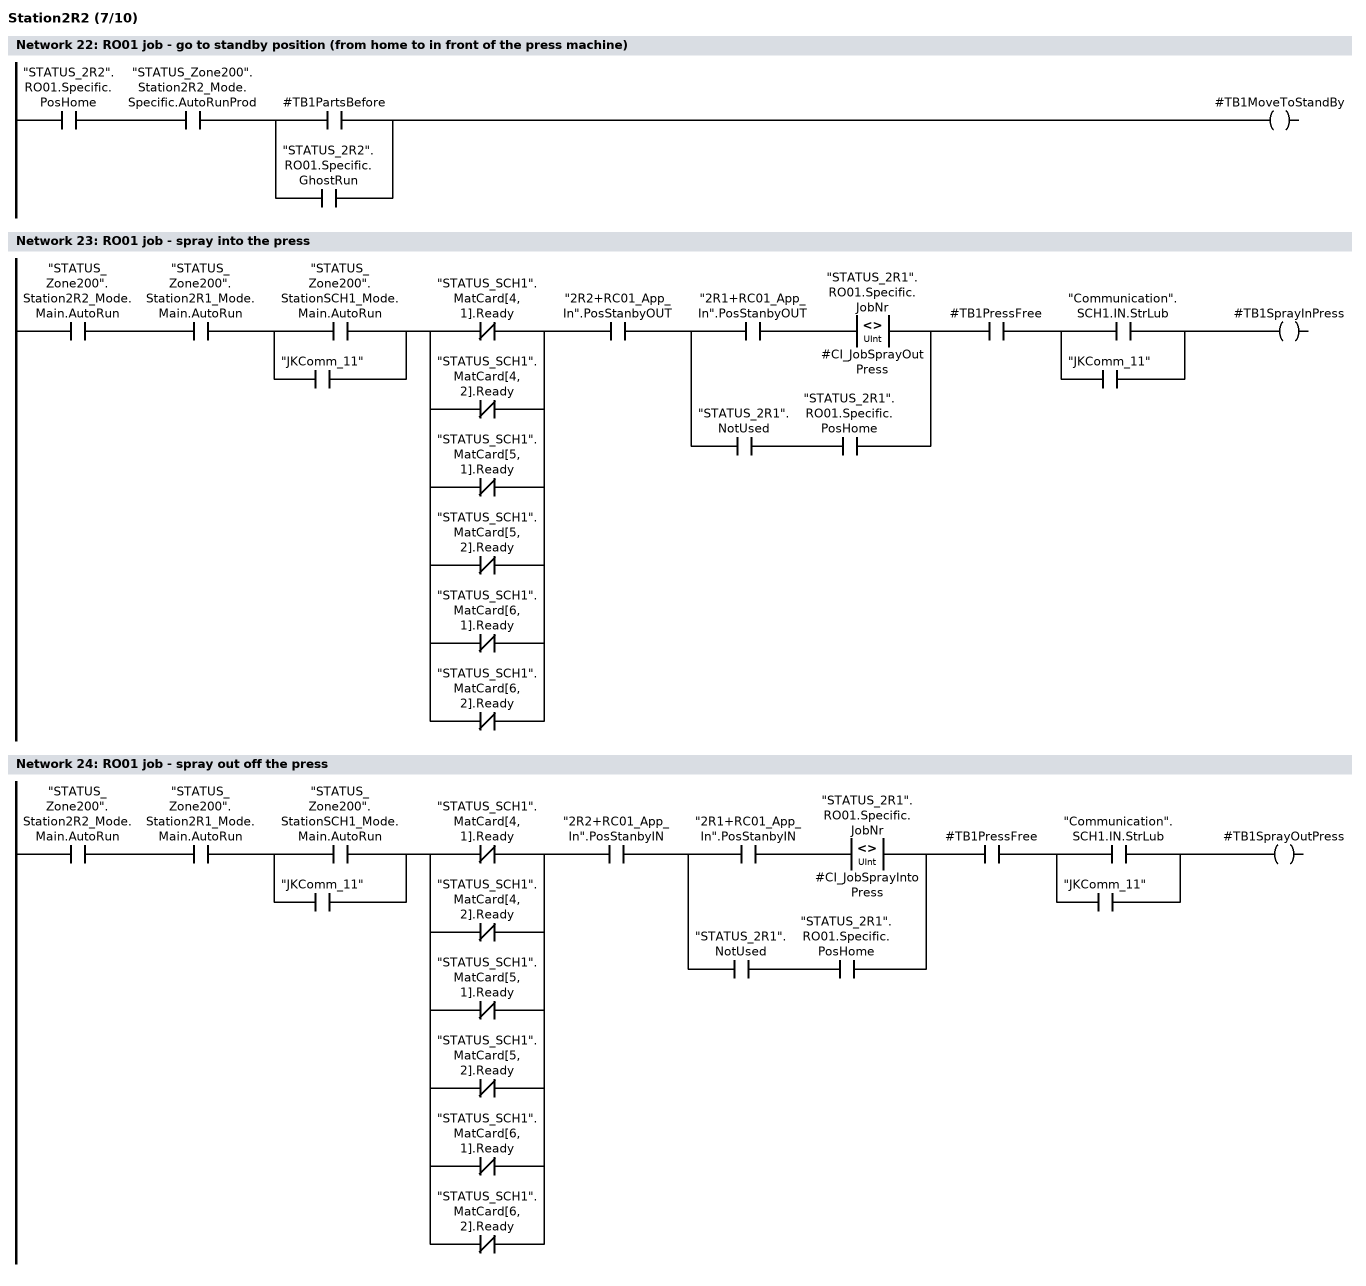
   RUNG wire#powerrail
      Contact( "STATUS_2R2".RO01.Specific.PosHome )
      Contact( "STATUS_Zone200".Station2R2_Mode.Specific.AutoRunProd )
      wire#w1
      Contact( #TB1PartsBefore )
      wire#w2
      Coil( #TB1MoveToStandBy )
   END_RUNG
   RUNG wire#w1
      Contact( "STATUS_2R2".RO01.Specific.GhostRun )
   END_RUNG wire#w2
   // the same network as SCL:
   #TB1MoveToStandBy := "STATUS_2R2".RO01.Specific.PosHome AND "STATUS_Zone200".Station2R2_Mode.Specific.AutoRunProd AND (#TB1PartsBefore OR "STATUS_2R2".RO01.Specific.GhostRun);
END_REGION

REGION Network 23: RO01 job - spray into the press
   RUNG wire#powerrail
      Contact( "STATUS_Zone200".Station2R2_Mode.Main.AutoRun )
      Contact( "STATUS_Zone200".Station2R1_Mode.Main.AutoRun )
      wire#w1
      Contact( "STATUS_Zone200".StationSCH1_Mode.Main.AutoRun )
      wire#w2
      I_Contact( "STATUS_SCH1".MatCard[4, 1].Ready )
      wire#w3
      Contact( "2R2+RC01_App_In".PosStanbyOUT )
      wire#w4
      Contact( "2R1+RC01_App_In".PosStanbyOUT )
      { S7_Templates := "SrcType := UInt" } NE_Contact(in1 := "STATUS_2R1".RO01.Specific.JobNr, in2 := #CI_JobSprayOutPress)
      wire#w5
      Contact( #TB1PressFree )
      wire#w6
      Contact( "Communication".SCH1.IN.StrLub )
      wire#w7
      Coil( #TB1SprayInPress )
   END_RUNG
   RUNG wire#w1
      Contact( "JKComm_11" )
   END_RUNG wire#w2
   RUNG wire#w2
      I_Contact( "STATUS_SCH1".MatCard[4, 2].Ready )
   END_RUNG wire#w3
   RUNG wire#w2
      I_Contact( "STATUS_SCH1".MatCard[5, 1].Ready )
   END_RUNG wire#w3
   RUNG wire#w2
      I_Contact( "STATUS_SCH1".MatCard[5, 2].Ready )
   END_RUNG wire#w3
   RUNG wire#w2
      I_Contact( "STATUS_SCH1".MatCard[6, 1].Ready )
   END_RUNG wire#w3
   RUNG wire#w2
      I_Contact( "STATUS_SCH1".MatCard[6, 2].Ready )
   END_RUNG wire#w3
   RUNG wire#w4
      Contact( "STATUS_2R1".NotUsed )
      Contact( "STATUS_2R1".RO01.Specific.PosHome )
   END_RUNG wire#w5
   RUNG wire#w6
      Contact( "JKComm_11" )
   END_RUNG wire#w7
   // the same network as SCL:
   #TB1SprayInPress := "STATUS_Zone200".Station2R2_Mode.Main.AutoRun AND "STATUS_Zone200".Station2R1_Mode.Main.AutoRun AND ("STATUS_Zone200".StationSCH1_Mode.Main.AutoRun OR "JKComm_11") AND (NOT "STATUS_SCH1".MatCard[4, 1].Ready OR NOT "STATUS_SCH1".MatCard[4, 2].Ready OR NOT "STATUS_SCH1".MatCard[5, 1].Ready OR NOT "STATUS_SCH1".MatCard[5, 2].Ready OR NOT "STATUS_SCH1".MatCard[6, 1].Ready OR NOT "STATUS_SCH1".MatCard[6, 2].Ready) AND "2R2+RC01_App_In".PosStanbyOUT AND (("2R1+RC01_App_In".PosStanbyOUT AND ("STATUS_2R1".RO01.Specific.JobNr <> #CI_JobSprayOutPress)) OR ("STATUS_2R1".NotUsed AND "STATUS_2R1".RO01.Specific.PosHome)) AND #TB1PressFree AND ("Communication".SCH1.IN.StrLub OR "JKComm_11");
END_REGION

REGION Network 24: RO01 job - spray out off the press
   RUNG wire#powerrail
      Contact( "STATUS_Zone200".Station2R2_Mode.Main.AutoRun )
      Contact( "STATUS_Zone200".Station2R1_Mode.Main.AutoRun )
      wire#w1
      Contact( "STATUS_Zone200".StationSCH1_Mode.Main.AutoRun )
      wire#w2
      I_Contact( "STATUS_SCH1".MatCard[4, 1].Ready )
      wire#w3
      Contact( "2R2+RC01_App_In".PosStanbyIN )
      wire#w4
      Contact( "2R1+RC01_App_In".PosStanbyIN )
      { S7_Templates := "SrcType := UInt" } NE_Contact(in1 := "STATUS_2R1".RO01.Specific.JobNr, in2 := #CI_JobSprayIntoPress)
      wire#w5
      Contact( #TB1PressFree )
      wire#w6
      Contact( "Communication".SCH1.IN.StrLub )
      wire#w7
      Coil( #TB1SprayOutPress )
   END_RUNG
   RUNG wire#w1
      Contact( "JKComm_11" )
   END_RUNG wire#w2
   RUNG wire#w2
      I_Contact( "STATUS_SCH1".MatCard[4, 2].Ready )
   END_RUNG wire#w3
   RUNG wire#w2
      I_Contact( "STATUS_SCH1".MatCard[5, 1].Ready )
   END_RUNG wire#w3
   RUNG wire#w2
      I_Contact( "STATUS_SCH1".MatCard[5, 2].Ready )
   END_RUNG wire#w3
   RUNG wire#w2
      I_Contact( "STATUS_SCH1".MatCard[6, 1].Ready )
   END_RUNG wire#w3
   RUNG wire#w2
      I_Contact( "STATUS_SCH1".MatCard[6, 2].Ready )
   END_RUNG wire#w3
   RUNG wire#w4
      Contact( "STATUS_2R1".NotUsed )
      Contact( "STATUS_2R1".RO01.Specific.PosHome )
   END_RUNG wire#w5
   RUNG wire#w6
      Contact( "JKComm_11" )
   END_RUNG wire#w7
   // the same network as SCL:
   #TB1SprayOutPress := "STATUS_Zone200".Station2R2_Mode.Main.AutoRun AND "STATUS_Zone200".Station2R1_Mode.Main.AutoRun AND ("STATUS_Zone200".StationSCH1_Mode.Main.AutoRun OR "JKComm_11") AND (NOT "STATUS_SCH1".MatCard[4, 1].Ready OR NOT "STATUS_SCH1".MatCard[4, 2].Ready OR NOT "STATUS_SCH1".MatCard[5, 1].Ready OR NOT "STATUS_SCH1".MatCard[5, 2].Ready OR NOT "STATUS_SCH1".MatCard[6, 1].Ready OR NOT "STATUS_SCH1".MatCard[6, 2].Ready) AND "2R2+RC01_App_In".PosStanbyIN AND (("2R1+RC01_App_In".PosStanbyIN AND ("STATUS_2R1".RO01.Specific.JobNr <> #CI_JobSprayIntoPress)) OR ("STATUS_2R1".NotUsed AND "STATUS_2R1".RO01.Specific.PosHome)) AND #TB1PressFree AND ("Communication".SCH1.IN.StrLub OR "JKComm_11");
END_REGION

REGION Network 25: RO01 - request to spray manual
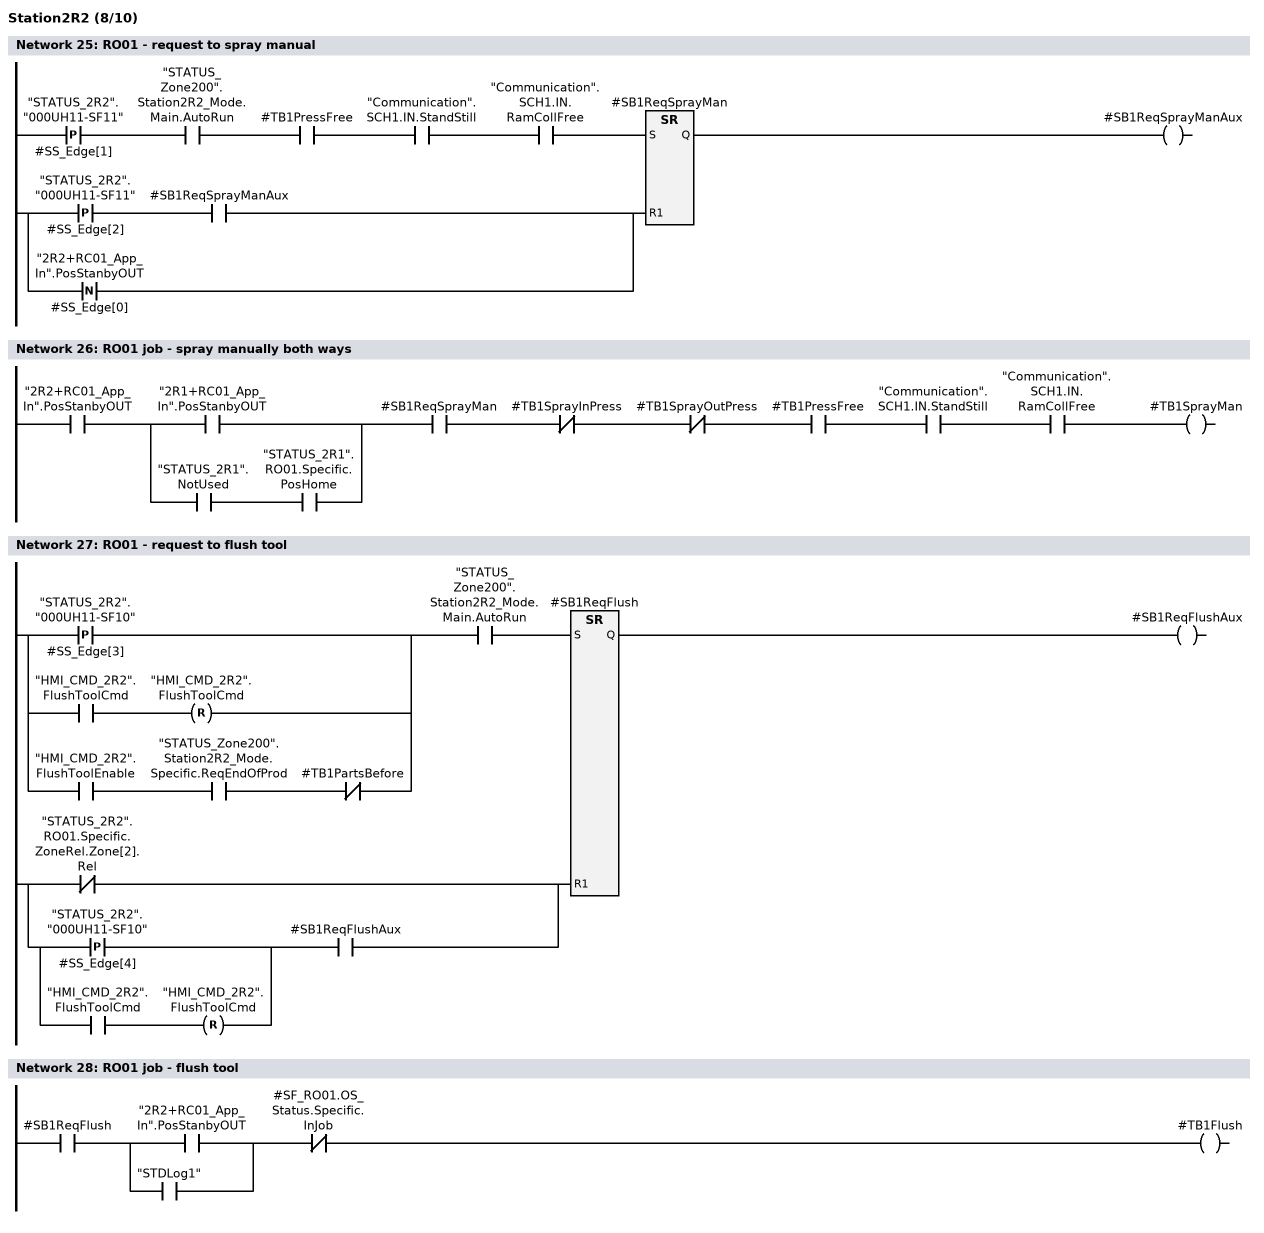
   RUNG wire#powerrail
      P_Contact(operand := "STATUS_2R2"."000UH11-SF11", bit := #SS_Edge[1])
      Contact( "STATUS_Zone200".Station2R2_Mode.Main.AutoRun )
      Contact( #TB1PressFree )
      Contact( "Communication".SCH1.IN.StandStill )
      Contact( "Communication".SCH1.IN.RamCollFree )
      S_SR(operand := #SB1ReqSprayMan, r1 := wire#w1)
      Coil( #SB1ReqSprayManAux )
   END_RUNG
   RUNG wire#powerrail
      P_Contact(operand := "STATUS_2R2"."000UH11-SF11", bit := #SS_Edge[2])
      Contact( #SB1ReqSprayManAux )
   END_RUNG wire#w1
   RUNG wire#powerrail
      N_Contact(operand := "2R2+RC01_App_In".PosStanbyOUT, bit := #SS_Edge[0])
   END_RUNG wire#w1
   // the same network as SCL:
   #_w1 := "STATUS_2R2"."000UH11-SF11" AND NOT #SS_Edge[1];   // rising edge of "STATUS_2R2"."000UH11-SF11"
   #SS_Edge[1] := "STATUS_2R2"."000UH11-SF11";
   #_w2 := "STATUS_2R2"."000UH11-SF11" AND NOT #SS_Edge[2];   // rising edge of "STATUS_2R2"."000UH11-SF11"
   #SS_Edge[2] := "STATUS_2R2"."000UH11-SF11";
   #_w3 := NOT "2R2+RC01_App_In".PosStanbyOUT AND #SS_Edge[0];   // falling edge of "2R2+RC01_App_In".PosStanbyOUT
   #SS_Edge[0] := "2R2+RC01_App_In".PosStanbyOUT;
   IF #_w1 AND "STATUS_Zone200".Station2R2_Mode.Main.AutoRun AND #TB1PressFree AND "Communication".SCH1.IN.StandStill AND "Communication".SCH1.IN.RamCollFree THEN
       #SB1ReqSprayMan := TRUE;   // SR flip-flop
   END_IF;
   IF (#_w2 AND #SB1ReqSprayManAux) OR #_w3 THEN #SB1ReqSprayMan := FALSE; END_IF;
   #SB1ReqSprayManAux := #SB1ReqSprayMan;
END_REGION

REGION Network 26: RO01 job - spray manually both ways
   RUNG wire#powerrail
      Contact( "2R2+RC01_App_In".PosStanbyOUT )
      wire#w1
      Contact( "2R1+RC01_App_In".PosStanbyOUT )
      wire#w2
      Contact( #SB1ReqSprayMan )
      I_Contact( #TB1SprayInPress )
      I_Contact( #TB1SprayOutPress )
      Contact( #TB1PressFree )
      Contact( "Communication".SCH1.IN.StandStill )
      Contact( "Communication".SCH1.IN.RamCollFree )
      Coil( #TB1SprayMan )
   END_RUNG
   RUNG wire#w1
      Contact( "STATUS_2R1".NotUsed )
      Contact( "STATUS_2R1".RO01.Specific.PosHome )
   END_RUNG wire#w2
   // the same network as SCL:
   #TB1SprayMan := "2R2+RC01_App_In".PosStanbyOUT AND ("2R1+RC01_App_In".PosStanbyOUT OR ("STATUS_2R1".NotUsed AND "STATUS_2R1".RO01.Specific.PosHome)) AND #SB1ReqSprayMan AND NOT #TB1SprayInPress AND NOT #TB1SprayOutPress AND #TB1PressFree AND "Communication".SCH1.IN.StandStill AND "Communication".SCH1.IN.RamCollFree;
END_REGION

REGION Network 27: RO01 - request to flush tool
   RUNG wire#powerrail
      P_Contact(operand := "STATUS_2R2"."000UH11-SF10", bit := #SS_Edge[3])
      wire#w1
      Contact( "STATUS_Zone200".Station2R2_Mode.Main.AutoRun )
      S_SR(operand := #SB1ReqFlush, r1 := wire#w3)
      Coil( #SB1ReqFlushAux )
   END_RUNG
   RUNG wire#powerrail
      Contact( "HMI_CMD_2R2".FlushToolCmd )
      R_Coil( "HMI_CMD_2R2".FlushToolCmd )
   END_RUNG wire#w1
   RUNG wire#powerrail
      Contact( "HMI_CMD_2R2".FlushToolEnable )
      Contact( "STATUS_Zone200".Station2R2_Mode.Specific.ReqEndOfProd )
      I_Contact( #TB1PartsBefore )
   END_RUNG wire#w1
   RUNG wire#powerrail
      I_Contact( "STATUS_2R2".RO01.Specific.ZoneRel.Zone[2].Rel )
   END_RUNG wire#w3
   RUNG wire#powerrail
      P_Contact(operand := "STATUS_2R2"."000UH11-SF10", bit := #SS_Edge[4])
      wire#w2
      Contact( #SB1ReqFlushAux )
   END_RUNG wire#w3
   RUNG wire#powerrail
      Contact( "HMI_CMD_2R2".FlushToolCmd )
      R_Coil( "HMI_CMD_2R2".FlushToolCmd )
   END_RUNG wire#w2
   // the same network as SCL:
   #_w1 := "STATUS_2R2"."000UH11-SF10" AND NOT #SS_Edge[3];   // rising edge of "STATUS_2R2"."000UH11-SF10"
   #SS_Edge[3] := "STATUS_2R2"."000UH11-SF10";
   #_w2 := "HMI_CMD_2R2".FlushToolCmd;
   IF #_w2 THEN "HMI_CMD_2R2".FlushToolCmd := FALSE; END_IF;
   #_w3 := "STATUS_2R2"."000UH11-SF10" AND NOT #SS_Edge[4];   // rising edge of "STATUS_2R2"."000UH11-SF10"
   #SS_Edge[4] := "STATUS_2R2"."000UH11-SF10";
   #_w4 := "HMI_CMD_2R2".FlushToolCmd;
   IF #_w4 THEN "HMI_CMD_2R2".FlushToolCmd := FALSE; END_IF;
   IF (#_w1 OR #_w2 OR ("HMI_CMD_2R2".FlushToolEnable AND "STATUS_Zone200".Station2R2_Mode.Specific.ReqEndOfProd AND NOT #TB1PartsBefore)) AND "STATUS_Zone200".Station2R2_Mode.Main.AutoRun THEN
       #SB1ReqFlush := TRUE;   // SR flip-flop
   END_IF;
   IF NOT "STATUS_2R2".RO01.Specific.ZoneRel.Zone[2].Rel OR ((#_w3 OR #_w4) AND #SB1ReqFlushAux) THEN
       #SB1ReqFlush := FALSE;
   END_IF;
   #SB1ReqFlushAux := #SB1ReqFlush;
END_REGION

REGION Network 28: RO01 job - flush tool
   RUNG wire#powerrail
      Contact( #SB1ReqFlush )
      wire#w1
      Contact( "2R2+RC01_App_In".PosStanbyOUT )
      wire#w2
      I_Contact( #SF_RO01.OS_Status.Specific.InJob )
      Coil( #TB1Flush )
   END_RUNG
   RUNG wire#w1
      Contact( "STDLog1" )
   END_RUNG wire#w2
   // the same network as SCL:
   #TB1Flush := #SB1ReqFlush AND ("2R2+RC01_App_In".PosStanbyOUT OR "STDLog1") AND NOT #SF_RO01.OS_Status.Specific.InJob;
END_REGION

REGION Network 29: RO01 job - move out off press
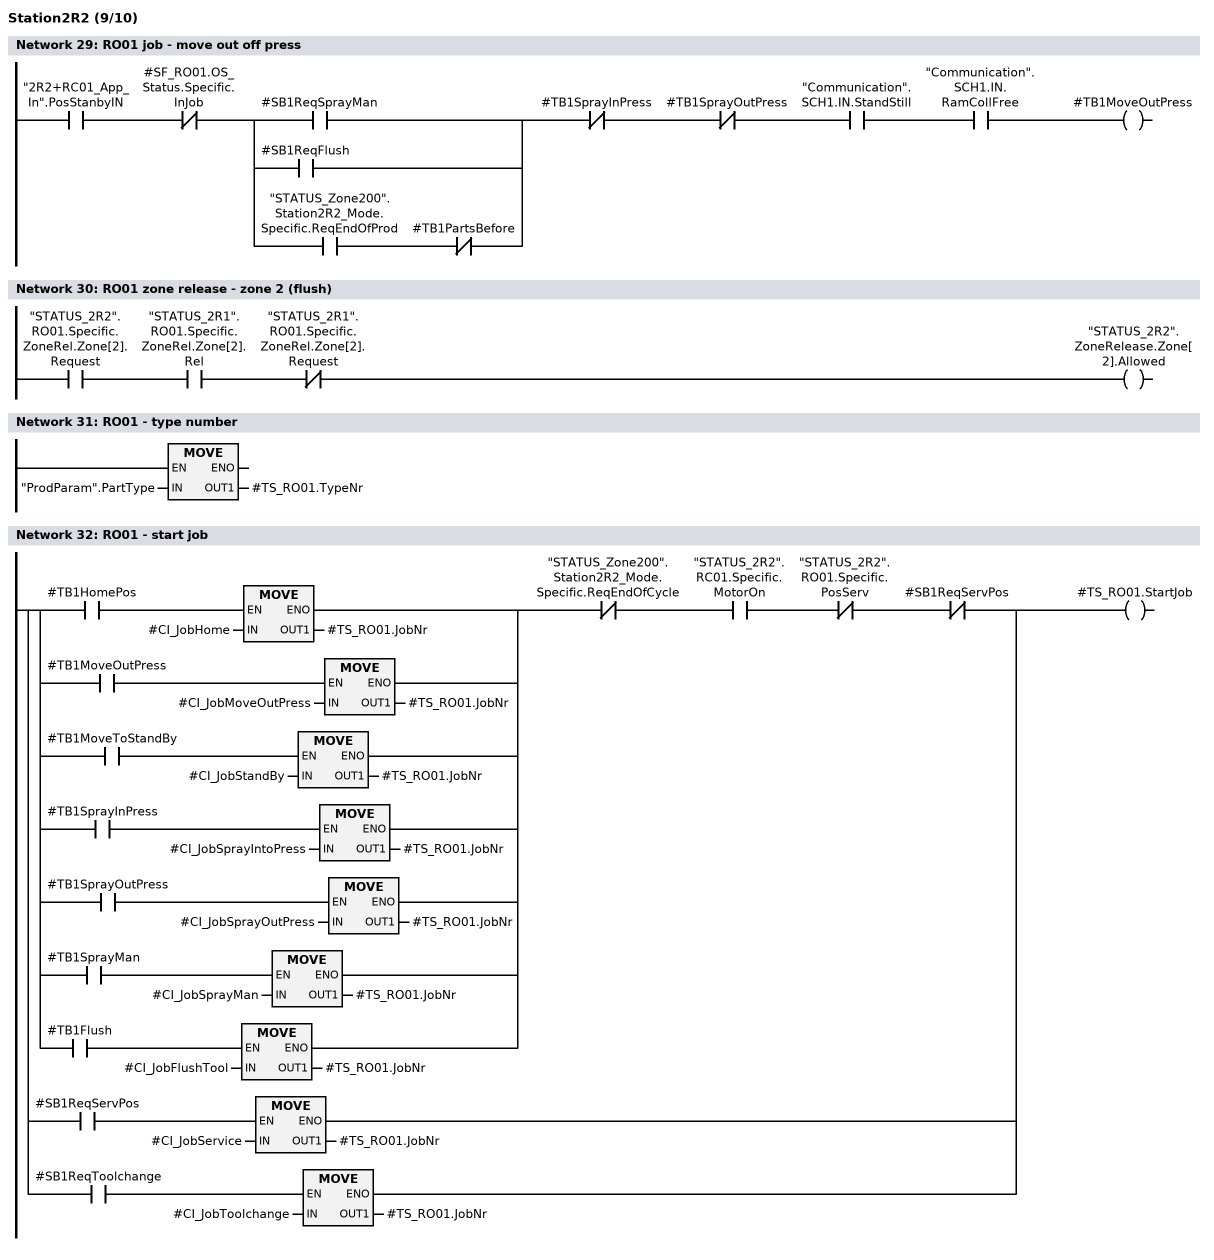
   RUNG wire#powerrail
      Contact( "2R2+RC01_App_In".PosStanbyIN )
      I_Contact( #SF_RO01.OS_Status.Specific.InJob )
      wire#w1
      Contact( #SB1ReqSprayMan )
      wire#w2
      I_Contact( #TB1SprayInPress )
      I_Contact( #TB1SprayOutPress )
      Contact( "Communication".SCH1.IN.StandStill )
      Contact( "Communication".SCH1.IN.RamCollFree )
      Coil( #TB1MoveOutPress )
   END_RUNG
   RUNG wire#w1
      Contact( #SB1ReqFlush )
   END_RUNG wire#w2
   RUNG wire#w1
      Contact( "STATUS_Zone200".Station2R2_Mode.Specific.ReqEndOfProd )
      I_Contact( #TB1PartsBefore )
   END_RUNG wire#w2
   // the same network as SCL:
   #TB1MoveOutPress := "2R2+RC01_App_In".PosStanbyIN AND NOT #SF_RO01.OS_Status.Specific.InJob AND (#SB1ReqSprayMan OR #SB1ReqFlush OR ("STATUS_Zone200".Station2R2_Mode.Specific.ReqEndOfProd AND NOT #TB1PartsBefore)) AND NOT #TB1SprayInPress AND NOT #TB1SprayOutPress AND "Communication".SCH1.IN.StandStill AND "Communication".SCH1.IN.RamCollFree;
END_REGION

REGION Network 30: RO01 zone release - zone 2 (flush)
   RUNG wire#powerrail
      Contact( "STATUS_2R2".RO01.Specific.ZoneRel.Zone[2].Request )
      Contact( "STATUS_2R1".RO01.Specific.ZoneRel.Zone[2].Rel )
      I_Contact( "STATUS_2R1".RO01.Specific.ZoneRel.Zone[2].Request )
      Coil( "STATUS_2R2".ZoneRelease.Zone[2].Allowed )
   END_RUNG
   // the same network as SCL:
   "STATUS_2R2".ZoneRelease.Zone[2].Allowed := "STATUS_2R2".RO01.Specific.ZoneRel.Zone[2].Request AND "STATUS_2R1".RO01.Specific.ZoneRel.Zone[2].Rel AND NOT "STATUS_2R1".RO01.Specific.ZoneRel.Zone[2].Request;
END_REGION

REGION Network 31: RO01 - type number
   RUNG wire#powerrail
      Move(in := "ProdParam".PartType, out1 => #TS_RO01.TypeNr)
   END_RUNG
   // the same network as SCL:
   #TS_RO01.TypeNr := "ProdParam".PartType;
END_REGION

REGION Network 32: RO01 - start job
   RUNG wire#powerrail
      Contact( #TB1HomePos )
      Move(in := #CI_JobHome, out1 => #TS_RO01.JobNr)
      wire#w1
      I_Contact( "STATUS_Zone200".Station2R2_Mode.Specific.ReqEndOfCycle )
      Contact( "STATUS_2R2".RC01.Specific.MotorOn )
      I_Contact( "STATUS_2R2".RO01.Specific.PosServ )
      I_Contact( #SB1ReqServPos )
      wire#w2
      Coil( #TS_RO01.StartJob )
   END_RUNG
   RUNG wire#powerrail
      Contact( #TB1MoveOutPress )
      Move(in := #CI_JobMoveOutPress, out1 => #TS_RO01.JobNr)
   END_RUNG wire#w1
   RUNG wire#powerrail
      Contact( #TB1MoveToStandBy )
      Move(in := #CI_JobStandBy, out1 => #TS_RO01.JobNr)
   END_RUNG wire#w1
   RUNG wire#powerrail
      Contact( #TB1SprayInPress )
      Move(in := #CI_JobSprayIntoPress, out1 => #TS_RO01.JobNr)
   END_RUNG wire#w1
   RUNG wire#powerrail
      Contact( #TB1SprayOutPress )
      Move(in := #CI_JobSprayOutPress, out1 => #TS_RO01.JobNr)
   END_RUNG wire#w1
   RUNG wire#powerrail
      Contact( #TB1SprayMan )
      Move(in := #CI_JobSprayMan, out1 => #TS_RO01.JobNr)
   END_RUNG wire#w1
   RUNG wire#powerrail
      Contact( #TB1Flush )
      Move(in := #CI_JobFlushTool, out1 => #TS_RO01.JobNr)
   END_RUNG wire#w1
   RUNG wire#powerrail
      Contact( #SB1ReqServPos )
      Move(in := #CI_JobService, out1 => #TS_RO01.JobNr)
   END_RUNG wire#w2
   RUNG wire#powerrail
      Contact( #SB1ReqToolchange )
      Move(in := #CI_JobToolchange, out1 => #TS_RO01.JobNr)
   END_RUNG wire#w2
   // the same network as SCL:
   IF #TB1HomePos THEN #TS_RO01.JobNr := #CI_JobHome; END_IF;
   IF #TB1MoveOutPress THEN #TS_RO01.JobNr := #CI_JobMoveOutPress; END_IF;
   IF #TB1MoveToStandBy THEN #TS_RO01.JobNr := #CI_JobStandBy; END_IF;
   IF #TB1SprayInPress THEN #TS_RO01.JobNr := #CI_JobSprayIntoPress; END_IF;
   IF #TB1SprayOutPress THEN #TS_RO01.JobNr := #CI_JobSprayOutPress; END_IF;
   IF #TB1SprayMan THEN #TS_RO01.JobNr := #CI_JobSprayMan; END_IF;
   IF #TB1Flush THEN #TS_RO01.JobNr := #CI_JobFlushTool; END_IF;
   IF #SB1ReqServPos THEN #TS_RO01.JobNr := #CI_JobService; END_IF;
   IF #SB1ReqToolchange THEN #TS_RO01.JobNr := #CI_JobToolchange; END_IF;
   #TS_RO01.StartJob := ((#TB1HomePos OR #TB1MoveOutPress OR #TB1MoveToStandBy OR #TB1SprayInPress OR #TB1SprayOutPress OR #TB1SprayMan OR #TB1Flush) AND NOT "STATUS_Zone200".Station2R2_Mode.Specific.ReqEndOfCycle AND "STATUS_2R2".RC01.Specific.MotorOn AND NOT "STATUS_2R2".RO01.Specific.PosServ AND NOT #SB1ReqServPos) OR #SB1ReqServPos OR #SB1ReqToolchange;
END_REGION

REGION Network 33: RO01 - main control (STD_RobotABB block call)
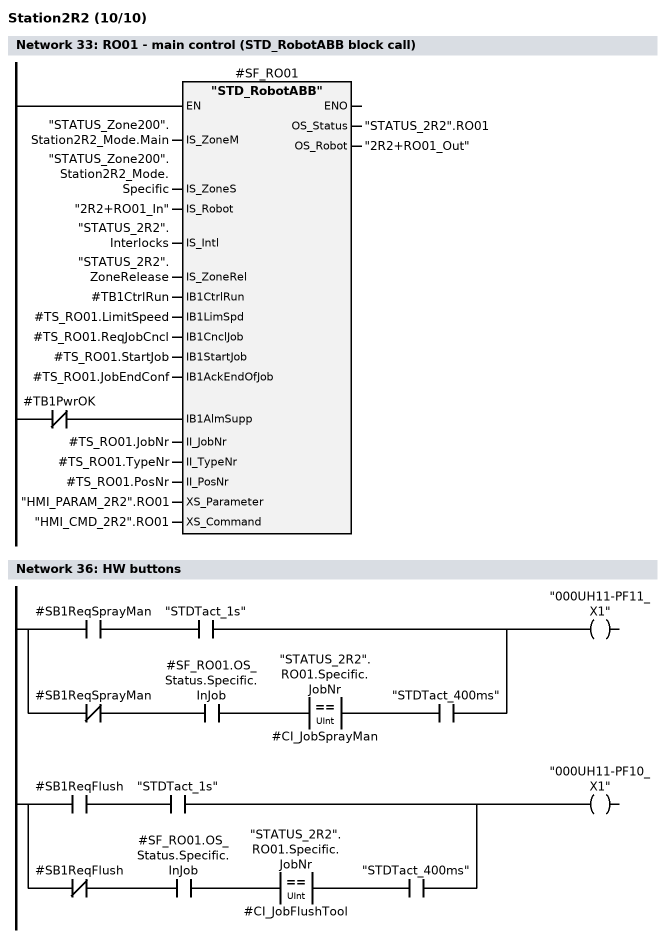
   RUNG wire#powerrail
      #SF_RO01(IB1AlmSupp := wire#w1, IS_ZoneM := "STATUS_Zone200".Station2R2_Mode.Main, IS_ZoneS := "STATUS_Zone200".Station2R2_Mode.Specific, IS_Robot := "2R2+RO01_In", IS_Intl := "STATUS_2R2".Interlocks, IS_ZoneRel := "STATUS_2R2".ZoneRelease, IB1CtrlRun := #TB1CtrlRun, IB1LimSpd := #TS_RO01.LimitSpeed, IB1CnclJob := #TS_RO01.ReqJobCncl, IB1StartJob := #TS_RO01.StartJob, IB1AckEndOfJob := #TS_RO01.JobEndConf, II_JobNr := #TS_RO01.JobNr, II_TypeNr := #TS_RO01.TypeNr, II_PosNr := #TS_RO01.PosNr, XS_Parameter := "HMI_PARAM_2R2".RO01, XS_Command := "HMI_CMD_2R2".RO01, OS_Status => "STATUS_2R2".RO01, OS_Robot => "2R2+RO01_Out")
   END_RUNG
   RUNG wire#powerrail
      I_Contact( #TB1PwrOK )
   END_RUNG wire#w1
   // the same network as SCL:
   #SF_RO01(IS_ZoneM := "STATUS_Zone200".Station2R2_Mode.Main,   // "STD_RobotABB"
            IS_ZoneS := "STATUS_Zone200".Station2R2_Mode.Specific,
            IS_Robot := "2R2+RO01_In",
            IS_Intl := "STATUS_2R2".Interlocks,
            IS_ZoneRel := "STATUS_2R2".ZoneRelease,
            IB1CtrlRun := #TB1CtrlRun,
            IB1LimSpd := #TS_RO01.LimitSpeed,
            IB1CnclJob := #TS_RO01.ReqJobCncl,
            IB1StartJob := #TS_RO01.StartJob,
            IB1AckEndOfJob := #TS_RO01.JobEndConf,
            IB1AlmSupp := NOT #TB1PwrOK,
            II_JobNr := #TS_RO01.JobNr,
            II_TypeNr := #TS_RO01.TypeNr,
            II_PosNr := #TS_RO01.PosNr,
            XS_Parameter := "HMI_PARAM_2R2".RO01,
            XS_Command := "HMI_CMD_2R2".RO01,
            OS_Status => "STATUS_2R2".RO01,
            OS_Robot => "2R2+RO01_Out");
END_REGION

REGION Network 34: ***************Aplication Interface***************
END_REGION

REGION Network 35: *************** Signalization ***************
END_REGION

REGION Network 36: HW buttons
   RUNG wire#powerrail
      Contact( #SB1ReqSprayMan )
      Contact( "STDTact_1s" )
      wire#w1
      Coil( "000UH11-PF11_X1" )
   END_RUNG
   RUNG wire#powerrail
      I_Contact( #SB1ReqSprayMan )
      Contact( #SF_RO01.OS_Status.Specific.InJob )
      { S7_Templates := "SrcType := UInt" } EQ_Contact(in1 := "STATUS_2R2".RO01.Specific.JobNr, in2 := #CI_JobSprayMan)
      Contact( "STDTact_400ms" )
   END_RUNG wire#w1
   RUNG wire#powerrail
      Contact( #SB1ReqFlush )
      Contact( "STDTact_1s" )
      wire#w2
      Coil( "000UH11-PF10_X1" )
   END_RUNG
   RUNG wire#powerrail
      I_Contact( #SB1ReqFlush )
      Contact( #SF_RO01.OS_Status.Specific.InJob )
      { S7_Templates := "SrcType := UInt" } EQ_Contact(in1 := "STATUS_2R2".RO01.Specific.JobNr, in2 := #CI_JobFlushTool)
      Contact( "STDTact_400ms" )
   END_RUNG wire#w2
   // the same network as SCL:
   "000UH11-PF11_X1" := (#SB1ReqSprayMan AND "STDTact_1s") OR (NOT #SB1ReqSprayMan AND #SF_RO01.OS_Status.Specific.InJob AND ("STATUS_2R2".RO01.Specific.JobNr = #CI_JobSprayMan) AND "STDTact_400ms");
   "000UH11-PF10_X1" := (#SB1ReqFlush AND "STDTact_1s") OR (NOT #SB1ReqFlush AND #SF_RO01.OS_Status.Specific.InJob AND ("STATUS_2R2".RO01.Specific.JobNr = #CI_JobFlushTool) AND "STDTact_400ms");
END_REGION
END_FUNCTION_BLOCK
